FUNCTION_BLOCK VCylinder (* Composite Function Block Type *)
  (* Standard: 61499-2 *)
  (* Version 0.0, 9/14/2008, Horst Mayer, nxtControl GmbH, template *)
  PACKAGE Main;
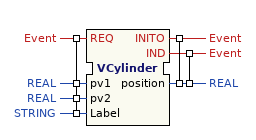
  EVENT_INPUT
    REQ WITH pv1, pv2, Label; (* Normal Execution Request *)
  END_EVENT
  EVENT_OUTPUT
    INITO WITH position;
    IND WITH position;
  END_EVENT
  VAR_INPUT
    pv1 : REAL;
    pv2 : REAL;
    Label : STRING;
  END_VAR
  VAR_OUTPUT
    position : REAL;
  END_VAR
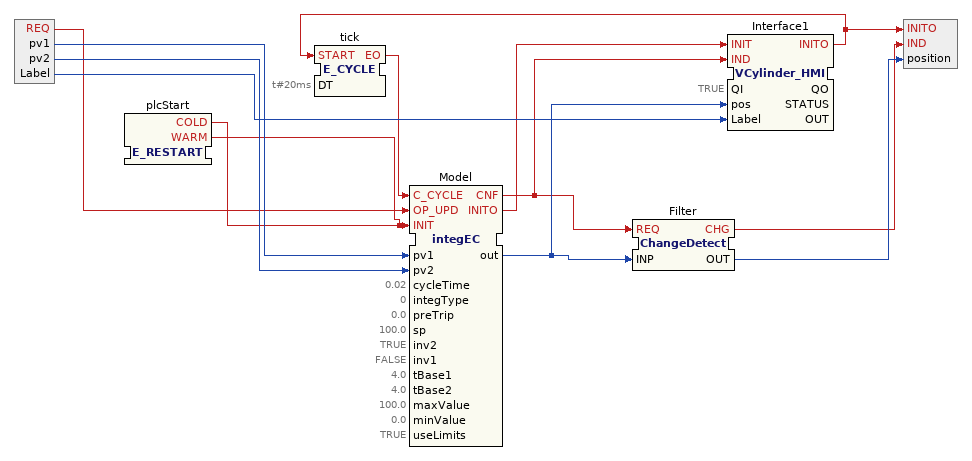
  FBS
    tick : E_CYCLE(DT := t#20ms);
    Interface1 : VCylinder_HMI(QI := TRUE);
    Model : integEC(cycleTime := 0.02, integType := 0, preTrip := 0.0, sp := 100.0, inv2 := TRUE, inv1 := FALSE, tBase1 := 4.0, tBase2 := 4.0, maxValue := 100.0, minValue := 0.0, useLimits := TRUE);
    plcStart : E_RESTART;
    Filter : ChangeDetect;
  END_FBS
  EVENT_CONNECTIONS
    Model.CNF TO Filter.REQ;
    tick.EO TO Model.C_CYCLE;
    REQ TO Model.OP_UPD;
    plcStart.COLD TO Model.INIT;
    plcStart.WARM TO Model.INIT;
    Filter.CHG TO IND;
    Model.INITO TO Interface1.INIT;
    Model.CNF TO Interface1.IND;
    Interface1.INITO TO tick.START;
    Interface1.INITO TO INITO;
  END_CONNECTIONS
  DATA_CONNECTIONS
    Model.out TO Filter.INP;
    pv1 TO Model.pv1;
    pv2 TO Model.pv2;
    Filter.OUT TO position;
    Model.out TO Interface1.pos;
    Label TO Interface1.Label;
  END_CONNECTIONS
END_FUNCTION_BLOCK
